PROGRAM controlejes
VAR
	MC_Power_eje1: MC_Power;
	MC_Power_eje2: MC_Power;
	MC_Stop_eje1: mc_stop;
	MC_Stop_eje2: mc_stop;
	MC_Reset_eje1: mc_reset;
	MC_Reset_eje2: mc_reset;
	MC_MoveAbsolute_eje1: MC_MoveAbsolute;
	MC_MoveAbsolute_eje2: MC_MoveAbsolute;
	
	MC_ReadStatus_eje1: MC_ReadStatus;
	MC_ReadStatus_eje2: MC_ReadStatus;
	
	MC_MoveVelocity_0: MC_MoveVelocity;
END_VAR

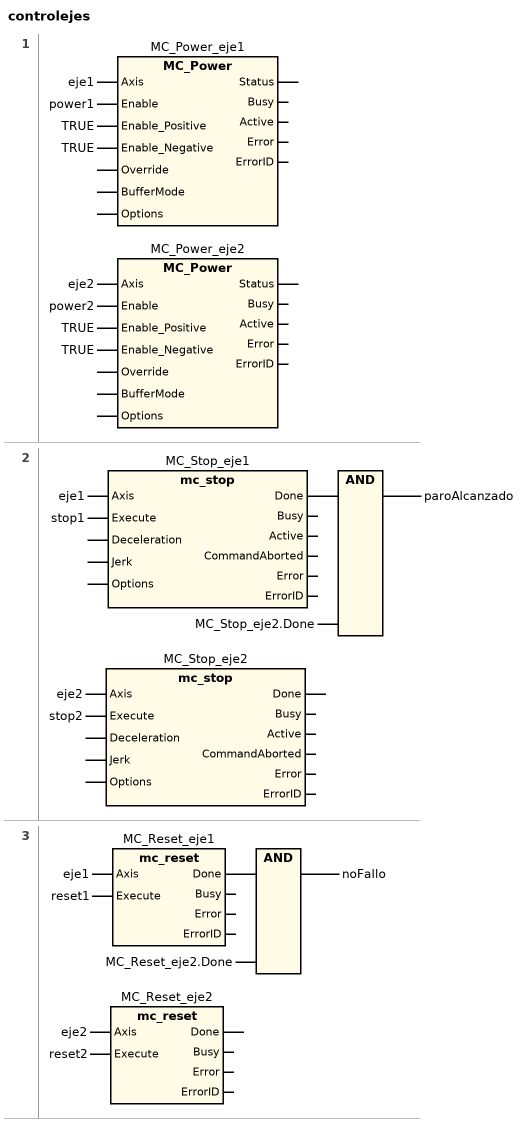
// NETWORK 1
MC_Power_eje1(Axis := eje1, Enable := power1, Enable_Positive := TRUE, Enable_Negative := TRUE); // MC_Power
MC_Power_eje2(Axis := eje2, Enable := power2, Enable_Positive := TRUE, Enable_Negative := TRUE); // MC_Power

// NETWORK 2
MC_Stop_eje1(Axis := eje1, Execute := stop1); // mc_stop
paroAlcanzado := MC_Stop_eje1.Done AND MC_Stop_eje2.Done;
MC_Stop_eje2(Axis := eje2, Execute := stop2); // mc_stop

// NETWORK 3
MC_Reset_eje1(Axis := eje1, Execute := reset1); // mc_reset
noFallo := MC_Reset_eje1.Done AND MC_Reset_eje2.Done;
MC_Reset_eje2(Axis := eje2, Execute := reset2); // mc_reset

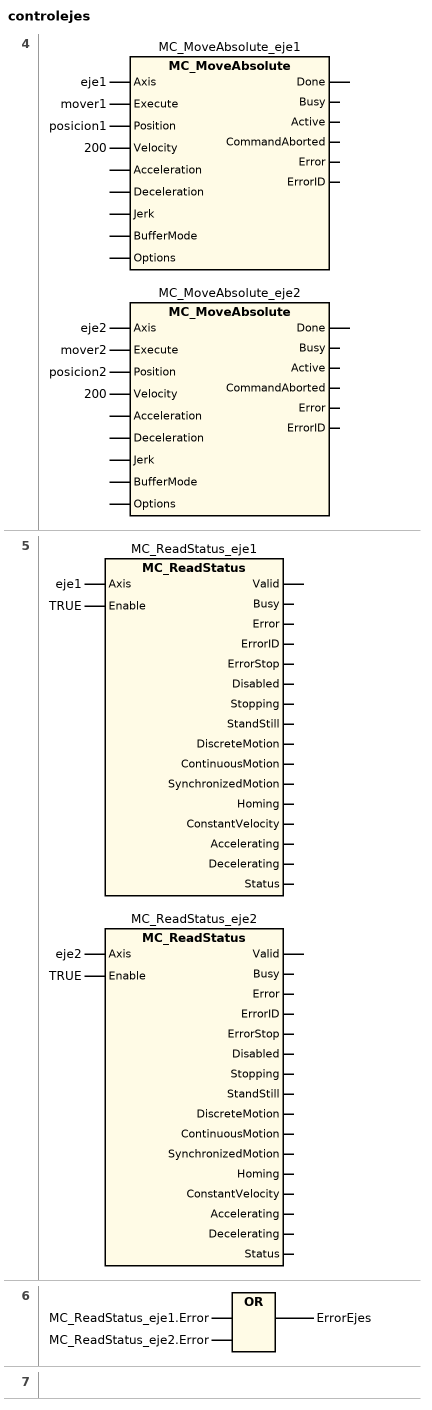
// NETWORK 4
MC_MoveAbsolute_eje1(Axis := eje1, Execute := mover1, Position := posicion1, Velocity := 200); // MC_MoveAbsolute
MC_MoveAbsolute_eje2(Axis := eje2, Execute := mover2, Position := posicion2, Velocity := 200); // MC_MoveAbsolute

// NETWORK 5
MC_ReadStatus_eje1(Axis := eje1, Enable := TRUE); // MC_ReadStatus
MC_ReadStatus_eje2(Axis := eje2, Enable := TRUE); // MC_ReadStatus

// NETWORK 6
ErrorEjes := MC_ReadStatus_eje1.Error OR MC_ReadStatus_eje2.Error;

// NETWORK 7

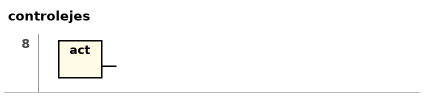
// NETWORK 8
act();

END_PROGRAM

(* stored: Version 1.1.0.1, ProductVersion 3.1.4024.9
   POU controlejes: Id {87198c64-e2f6-4075-ba4e-19df934b96c0}, SpecialFunc None *)
